{attribute 'GeneratedUsingTerminal: EL2535-0103-0023'}
{attribute addProperty BoxType "EL2535-0103-0023"}
{attribute addProperty Id "StatusAT %I*Status_72C27E804"}
{attribute addProperty CRC "2006162193"}
{attribute addProperty Size "4"}
TYPE PWM_Status_Channel_77939B11 EXTENDS InputBase_8311D824 :
STRUCT
	{attribute addProperty Name "Status"}
	Status AT %I* : Status_72C27E80;
END_STRUCT
END_TYPE

(* stored: Version 1.2.0.0, ProductVersion 3.1.4024.11
   DUT PWM_Status_Channel_77939B11: Id {bc82669c-00b9-4d66-aaad-4acd7b8e7300} *)
